PROGRAM ManualMode
VAR
	ABBFunction: INT;
	PickLeave: INT;
	BufferID: INT;
	Part: INT;

	Execute: BOOL;
	mxExecute: BOOL;
	
	AssebmleExecuting: BOOL;
	GotoAGVExecuting: BOOL;
	GotoBufferExecuting: BOOL;
	GotoHomeExecuting: BOOL;
	GotoScannerExecuting: BOOL;
	GotoTableExecuting: BOOL;
	PickLeaveBufferExecuting: BOOL;
	PickLeaveContainerExecuting: BOOL;
	PickLeaveContaineronTableExecuting: BOOL;
	PickLeaveScannerExecuting: BOOL;
	ScanContainerExecuting: BOOL;
	ScannerStationExecuting: BOOL;
	
	AssebmleError: BOOL;
	GotoAGVError: BOOL;
	GotoBufferError: BOOL;
	GotoHomeError: BOOL;
	GotoScannerError: BOOL;
	GotoTableError: BOOL;
	PickLeaveBufferError: BOOL;
	PickLeaveContainerError: BOOL;
	PickLeaveContaineronTableError: BOOL;
	PickLeaveScannerError: BOOL;
	ScanContainerError: BOOL;
	ScannerStationError: BOOL;
	
	ABBAssemble_Manual: ABBAssemble;
	ABBGotoAGVPos_Manual: ABBGotoAGVPos;
	ABBGotoBuffer_Manual: ABBGotoBuffer;
	ABBGotoHome_Manual: ABBGotoHome;
	ABBGotoScanner_Manual: ABBGotoScanner;
	ABBGotoTable_Manual: ABBGotoTable;
	ABBPickLeaveBuffer_Manual: ABBPickLeaveBuffer;
	ABBPickLeaveContainerAGV_Manual: ABBPickLeaveContainerAGV;
	ABBPickLeaveContaineronTable_Manual: ABBPickLeaveContaineronTable;
	ABBPickLeaveScanner_Manual: ABBPickLeaveScanner;
	ABBScanContainer_Manual: ABBScanContainer;
	ABBScannerStation_Manual: ABBScannerStation;
END_VAR

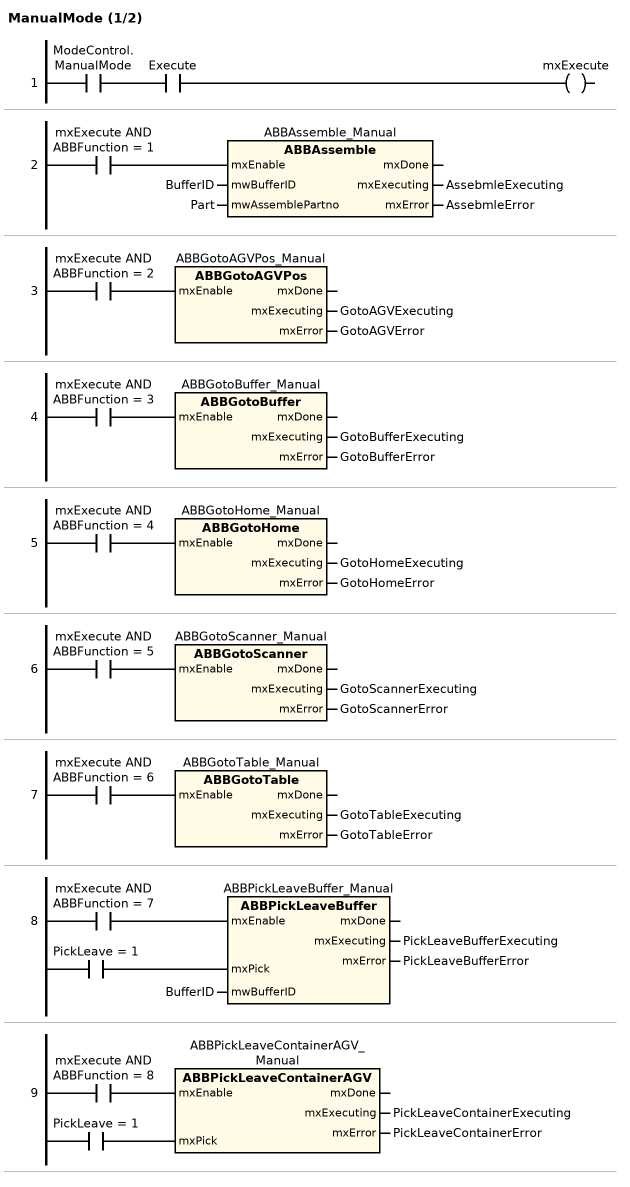
// NETWORK 1
mxExecute := ModeControl.ManualMode AND Execute;

// NETWORK 2
ABBAssemble_Manual(
    mxEnable := mxExecute AND ABBFunction = 1,
    mwBufferID := BufferID,
    mwAssemblePartno := Part,
    mxExecuting => AssebmleExecuting,
    mxError => AssebmleError); // ABBAssemble

// NETWORK 3
ABBGotoAGVPos_Manual(
    mxEnable := mxExecute AND ABBFunction = 2,
    mxExecuting => GotoAGVExecuting,
    mxError => GotoAGVError); // ABBGotoAGVPos

// NETWORK 4
ABBGotoBuffer_Manual(
    mxEnable := mxExecute AND ABBFunction = 3,
    mxExecuting => GotoBufferExecuting,
    mxError => GotoBufferError); // ABBGotoBuffer

// NETWORK 5
ABBGotoHome_Manual(
    mxEnable := mxExecute AND ABBFunction = 4,
    mxExecuting => GotoHomeExecuting,
    mxError => GotoHomeError); // ABBGotoHome

// NETWORK 6
ABBGotoScanner_Manual(
    mxEnable := mxExecute AND ABBFunction = 5,
    mxExecuting => GotoScannerExecuting,
    mxError => GotoScannerError); // ABBGotoScanner

// NETWORK 7
ABBGotoTable_Manual(
    mxEnable := mxExecute AND ABBFunction = 6,
    mxExecuting => GotoTableExecuting,
    mxError => GotoTableError); // ABBGotoTable

// NETWORK 8
ABBPickLeaveBuffer_Manual(
    mxEnable := mxExecute AND ABBFunction = 7,
    mxPick := PickLeave = 1,
    mwBufferID := BufferID,
    mxExecuting => PickLeaveBufferExecuting,
    mxError => PickLeaveBufferError); // ABBPickLeaveBuffer

// NETWORK 9
ABBPickLeaveContainerAGV_Manual(
    mxEnable := mxExecute AND ABBFunction = 8,
    mxPick := PickLeave = 1,
    mxExecuting => PickLeaveContainerExecuting,
    mxError => PickLeaveContainerError); // ABBPickLeaveContainerAGV

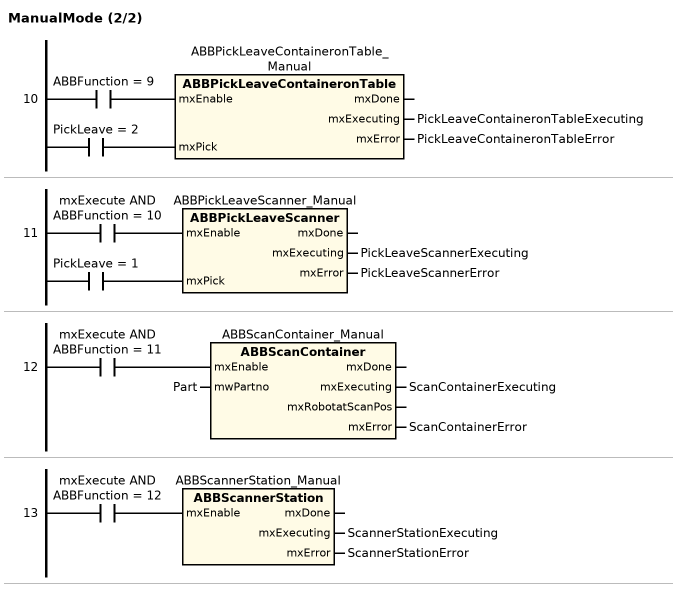
// NETWORK 10
ABBPickLeaveContaineronTable_Manual(
    mxEnable := ABBFunction = 9,
    mxPick := PickLeave = 2,
    mxExecuting => PickLeaveContaineronTableExecuting,
    mxError => PickLeaveContaineronTableError); // ABBPickLeaveContaineronTable

// NETWORK 11
ABBPickLeaveScanner_Manual(
    mxEnable := mxExecute AND ABBFunction = 10,
    mxPick := PickLeave = 1,
    mxExecuting => PickLeaveScannerExecuting,
    mxError => PickLeaveScannerError); // ABBPickLeaveScanner

// NETWORK 12
ABBScanContainer_Manual(
    mxEnable := mxExecute AND ABBFunction = 11,
    mwPartno := Part,
    mxExecuting => ScanContainerExecuting,
    mxError => ScanContainerError); // ABBScanContainer

// NETWORK 13
ABBScannerStation_Manual(
    mxEnable := mxExecute AND ABBFunction = 12,
    mxExecuting => ScannerStationExecuting,
    mxError => ScannerStationError); // ABBScannerStation

END_PROGRAM

(* stored: Version 1.1.0.1, ProductVersion 3.1.4024.12
   POU ManualMode: Id {21a62cce-8f3a-461e-b544-40bd6363776d}, SpecialFunc None *)
